// SIMATIC STEP 7 (V5.x) project PUERTA DB
// program: Programa S7(1)

DATA_BLOCK DB 1
//VARIABLES A NIVEL DE BIT
VERSION : 0.1
  STRUCT
   MARCA0 : BOOL ;
   MARCA1 : BOOL ;
   MARCA2 : BOOL ;
   MARCA3 : BOOL ;
   MARCA4 : BOOL ;
   MARCA5 : BOOL ;
   MARCA6 : BOOL ;
   MARCA7 : BOOL ;
   MARCA8 : BOOL ;
   MARCA9 : BOOL ;
  END_STRUCT ;	
BEGIN
END_DATA_BLOCK

ORGANIZATION_BLOCK OB 1
TITLE = "Main Program Sweep (Cycle)"
VERSION : 0.1
VAR_TEMP
  OB1_EV_CLASS : BYTE ;	//Bits 0-3 = 1 (Coming event), Bits 4-7 = 1 (Event class 1)
  OB1_SCAN_1 : BYTE ;	//1 (Cold restart scan 1 of OB 1), 3 (Scan 2-n of OB 1)
  OB1_PRIORITY : BYTE ;	//Priority of OB Execution
  OB1_OB_NUMBR : BYTE ;	//1 (Organization block 1, OB1)
  OB1_RESERVED_1 : BYTE ;	//Reserved for system
  OB1_RESERVED_2 : BYTE ;	//Reserved for system
  OB1_PREV_CYCLE : INT ;	//Cycle time of previous OB1 scan (milliseconds)
  OB1_MIN_CYCLE : INT ;	//Minimum cycle time of OB1 (milliseconds)
  OB1_MAX_CYCLE : INT ;	//Maximum cycle time of OB1 (milliseconds)
  OB1_DATE_TIME : DATE_AND_TIME ;	//Date and time OB1 started
END_VAR
BEGIN
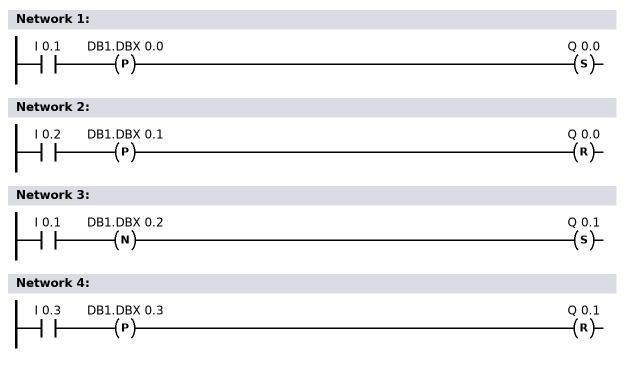
NETWORK
TITLE =
      A     I 0.1;
      FP    DB1.DBX 0.0;
      S     Q 0.0;
NETWORK
TITLE =
      A     I 0.2;
      FP    DB1.DBX 0.1;
      R     Q 0.0;
NETWORK
TITLE =
      A     I 0.1;
      FN    DB1.DBX 0.2;
      S     Q 0.1;
NETWORK
TITLE =
      A     I 0.3;
      FP    DB1.DBX 0.3;
      R     Q 0.1;
NETWORK
TITLE =
END_ORGANIZATION_BLOCK
